// Mitsubishi GX Works2 project: semaforo   PLC: Q03UDV

PROGRAM MAIN
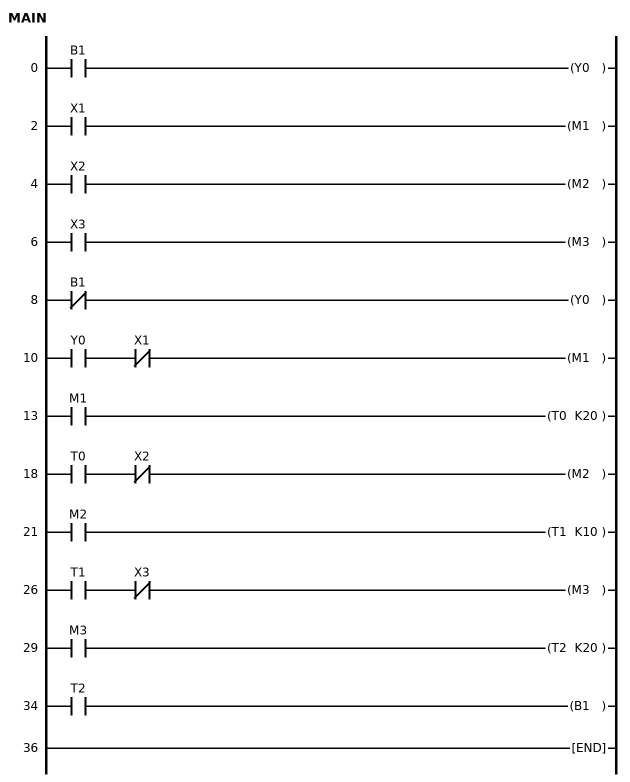
0     LD      B1
      OUT     Y0
2     LD      X1
      OUT     M1
4     LD      X2
      OUT     M2
6     LD      X3
      OUT     M3
8     LDI     B1
      OUT     Y0
10    LD      Y0
      ANI     X1
      OUT     M1
13    LD      M1
      OUT     T0 K20
18    LD      T0
      ANI     X2
      OUT     M2
21    LD      M2
      OUT     T1 K10
26    LD      T1
      ANI     X3
      OUT     M3
29    LD      M3
      OUT     T2 K20
34    LD      T2
      OUT     B1
36    END
END_PROGRAM
